// TIA Portal V20 export
FUNCTION_BLOCK "FB_ScannerComm"   // FB85, SCL
{ S7_Optimized_Access := 'TRUE' }
// stored: MemoryReserve 100, SetENOAutomatically false
   VAR_INPUT
      iInit : Bool;
      iReady : Bool;   // From HMI OPC UA
      iStatus : DInt;   // From HMI OPC UA
      iStatusDescription : String;   // From HMI OPC UA
      iCheckNumber : Byte;   // From HMI OPC UA
      iPartOnFixture : Bool;
      iStationNumber : Byte;   // From NC ?
      iHoleNumber : DInt;   // From NC ?
      iJobListName : String;   // From NC ?
      iJobName : DInt;   // From NC ?
      iMeasureZ : LReal;   // From NC ?
   END_VAR
   VAR_OUTPUT
      oIsFirstJobOfPiece : Bool;
      oStationNumber : Byte;
      oHoleNumber : DInt;
      oJobListName : String;
      oJobName : String;
      oMeasureZ : LReal;
      oBadPart : Bool;
      oGoodPart : Bool;
      oEndOfJob : Bool;
   END_VAR
   VAR_IN_OUT
      ioRequestJob_NC : Bool;   // From NC ?
      ioReady_NC : Bool;   // From NC ?
      ioCheckNumber : Byte;
      ioRequestJob : Bool;
   END_VAR
   VAR
      sRT_PartOnFixture : R_TRIG;
      sRT_Ready { S7_SetPoint := 'True'} : R_TRIG;
      sEndOfJob { S7_SetPoint := 'True'} : Bool;
      sRT_RequestJob_NC : R_TRIG;
      sJobListName { S7_SetPoint := 'True'} : String;
      sJobName : String;
      sJobInProgress : Bool;
   END_VAR
BEGIN
   REGION Description header 
       //==================================================================================
       // POSALUX Swiss SA / (C) Copyright 2026
       //----------------------------------------------------------------------------------
       // Title: FB_ScannerComm
       // Comment/Function: 
       //
       // Author: Fabien WALDT
       // Engineering: TIA Portal v20
       //----------------------------------------------------------------------------------
       // Change log table:
       // Version  | Date     | Expert in charge | Changes applied
       // ---------|----------|------------------|------------------------------------
       // 00.00.01 | 20260330 | WFA              | First released version
       // ==================================================================================
   END_REGION

   REGION R_Trig
       #sRT_PartOnFixture(CLK := #iPartOnFixture);

       #sRT_Ready(CLK := #iReady);
       #sEndOfJob := #sRT_Ready.Q AND #sJobInProgress;

       #sRT_RequestJob_NC(CLK := #ioRequestJob_NC);
   END_REGION

   REGION Job
   #sJobListName := #iJobListName;
   #sJobName := DINT_TO_STRING(IN := #iJobName);

   IF #sJobName[1] = '+' THEN
       #sJobName := DELETE(IN := #sJobName, L := 1, P := 1);
   END_IF;
   END_REGION

   REGION Parameters
       // IsFirstJobOfPiece 
       IF #sRT_PartOnFixture.Q THEN
           #oIsFirstJobOfPiece := TRUE;
       ELSIF #sEndOfJob OR NOT #iPartOnFixture THEN
           #oIsFirstJobOfPiece := FALSE;
       END_IF;

       IF #sRT_RequestJob_NC.Q THEN
           // StationNumber 
           #oStationNumber := #iStationNumber;

           // HoleNumber 
           #oHoleNumber := #iHoleNumber;

           // JobListName 
           #oJobListName := #sJobListName;

           // JobName 
           #oJobName := #sJobName;

           // MeasureZ 
           #oMeasureZ := #iMeasureZ;

           // CheckNumber Increment
           #ioCheckNumber := #ioCheckNumber + 1;
           IF #ioCheckNumber > 255 OR #ioCheckNumber < 1 THEN
               #ioCheckNumber := 1;
           END_IF;

           // Reset Bad/Good Part
           #oBadPart := FALSE;
           #oGoodPart := FALSE;
       END_IF;
   END_REGION

   REGION Request Job
       IF #ioRequestJob_NC AND #iReady AND NOT #sJobInProgress THEN
           #sJobInProgress := TRUE;
           #ioRequestJob := TRUE;
       ELSIF (#ioRequestJob AND NOT #iReady) OR #iInit THEN
           #ioRequestJob := FALSE;
       END_IF;
   END_REGION

   REGION End of Job
       IF #sEndOfJob THEN
           IF #ioCheckNumber = #iCheckNumber AND #iStatus = 1 THEN
               #oGoodPart := TRUE;
           ELSE
               #oBadPart := TRUE;
           END_IF;
           #sJobInProgress := FALSE;
       END_IF;

       // Update Output
       #oEndOfJob := #sEndOfJob;
   END_REGION
END_FUNCTION_BLOCK
